Omron Sysmac Studio project Foset_Youtube_jp (Sysmac Studio 1.54.0.64019, StandardProject)

# Controller new_Controller_0: NX102-1220 version 1.48
Units and slaves: Node10 : NX-ECC203 (E001); Unit 1 : NX-PF0630 (N2); Unit 2 : NX-ID4442 (N3); Unit 3 : NX-OD4256 (N4); Unit 4 : NX-ILM400 (N5); Unit 5 : NX-SID800 (N6); Unit 6 : NX-SOD400 (N7)
Task PrimaryTask (priority 4, period or condition 2000): Program0

TYPE Byte2Bool : UNION
    ByteData : BYTE;
    BoolData : ARRAY[0..7] OF bool;
END_UNION END_TYPE
TYPE Byte2Word : UNION
    ByteData : ARRAY[0..1] OF byte;
    WordData : WORD;
END_UNION END_TYPE
TYPE DUT_E3ASHL500MN_ProcessData_Byte3 : STRUCT
    ControlOutput1 : BOOL;
    ControlOutput2 : BOOL;
    LowIntensity : BOOL;
    IssficientLioghtIntensity : BOOL;
    Warning : BOOL;
    Error : BOOL;
END_STRUCT END_TYPE
TYPE DUT_E3ASHL500MN_ProcessData : STRUCT
    DetectionValue : INT;
    LightIntensity : INT;
    Status : DUT_E3ASHL500MN_ProcessData_Byte3;
END_STRUCT END_TYPE

VAR_GLOBAL
    N3_Input_Bit_8_bits : BYTE;  (* at ECAT://node#[10,2]/Input Bit 8 bits *)
    N4_Output_Bit_8_bits : BYTE;  (* at ECAT://node#[10,3]/Output Bit 8 bits *)
    N5_Port2_Input_Data01 : ARRAY[0..1] OF BYTE;  (* at ECAT://node#[10,4]/Port2 Input Data01 *)
    N5_Port2_Input_Data02 : ARRAY[0..1] OF BYTE;  (* at ECAT://node#[10,4]/Port2 Input Data02 *)
    N5_Port2_IN_Data_Enable : BOOL;  (* at ECAT://node#[10,4]/I/O Port Status/Port2 IN Data Enable *)
    N5_IO_Pwr_On : BOOL;  (* at ECAT://node#[10,4]/I/O Port Status/IO Pwr On *)
    N6_Si00_Logical_Value : BOOL;  (* at ECAT://node#[10,5]/Standard Input 1st Word/Si00 Logical Value *)
    N1_DataToSafety_01 : BOOL;  (* at IOBus://unit#1/DataToSafety_01 *)
    N1_DataToSafety_00 : BOOL;  (* at IOBus://unit#1/DataToSafety_00 *)
    N1_Program_Operating : BOOL;  (* at IOBus://unit#1/Program Operating *)
    N1_Program_No_Fault : BOOL;  (* at IOBus://unit#1/Program No Fault *)
    N1_CIP_Safety_Originator_Connection_Status : BOOL;  (* at IOBus://unit#1/CIP Safety Originator Connection Status *)
END_VAR

(* Program Program0: safety or other program stored in binary form, left out *)

PROGRAM Program0
VAR
    NodeReady : BOOL;
    bNoContact : BOOL;
    bNCContact : BOOL;
    MyTimer1 : TON;
    MyTimer2 : TON;
    MyTimer3 : TON;
    MyTimer4 : TON;
    strByte2Bool : Byte2Bool;
    E3AS_1 : FB_E3ASHL500MN;
    Device : DUT_E3ASHL500MN_ProcessData;
    Port2Ready : BOOL;
END_VAR
VAR_EXTERNAL
    N1_DataToSafety_01 : BOOL;
END_VAR
VAR_EXTERNAL CONSTANT
    _EC_MacAdrErr : BOOL;
    _EC_CommErrTbl : ARRAY[1..192] OF BOOL;
END_VAR
VAR_EXTERNAL
    N3_Input_Bit_8_bits : BYTE;
    N1_DataToSafety_00 : BOOL;
    N1_Program_No_Fault : BOOL;
    N1_CIP_Safety_Originator_Connection_Status : BOOL;
    N1_Program_Operating : BOOL;
    N6_Si00_Logical_Value : BOOL;
    N5_Port2_IN_Data_Enable : BOOL;
    N5_IO_Pwr_On : BOOL;
    N5_Port2_Input_Data01 : ARRAY[0..1] OF BYTE;
    N5_Port2_Input_Data02 : ARRAY[0..1] OF BYTE;
    N4_Output_Bit_8_bits : BYTE;
END_VAR
//
	MyTimer3(In:=NOT MyTimer4.Q, PT:=T#0.5s);
	MyTimer4(In:=MyTimer3.Q, PT:=T#0.5s);
	N1_DataToSafety_01:=MyTimer3.Q;
	
//
	NodeReady:=_EC_MacAdrErr = 0 AND NOT _EC_CommErrTbl[2];
	strByte2Bool.ByteData:=0;
	strByte2Bool.ByteData:=N3_Input_Bit_8_bits;
	bNoContact:=strByte2Bool.BoolData[0];
	bNCContact:=strByte2Bool.BoolData[1];
	N1_DataToSafety_00:=strByte2Bool.BoolData[2] AND 
			N1_Program_No_Fault AND N1_Program_Operating AND N6_Si00_Logical_Value;
//
	strByte2Bool.ByteData:=0;
	NodeReady:=_EC_MacAdrErr = 0 AND NOT _EC_CommErrTbl[3];
	MyTimer1(In:=bNoContact AND NOT MyTimer2.Q, PT:=T#1s);
	MyTimer2(In:=MyTimer1.Q, PT:=T#1s);
	strByte2Bool.BoolData[1]:=bNCContact OR MyTimer1.Q;
	N4_Output_Bit_8_bits:=strByte2Bool.ByteData;
	
//
	Port2Ready:=N5_Port2_IN_Data_Enable AND N5_IO_Pwr_On;
	NodeReady:=_EC_MacAdrErr = 0 AND NOT _EC_CommErrTbl[5];
	E3AS_1	(IoData1:=N5_Port2_Input_Data01,IoData2:=N5_Port2_Input_Data02
				,ioE3AS:=Device
				);
				
END_PROGRAM

FUNCTION_BLOCK FB_E3ASHL500MN
VAR
    Temp : BOOL;
    uByte2Word : Byte2Word;
    uByteBool : Byte2Bool;
END_VAR
VAR_IN_OUT
    ioData1 : ARRAY[0..1] OF byte;
    ioData2 : ARRAY[0..1] OF byte;
    ioE3AS : DUT_E3ASHL500MN_ProcessData;
END_VAR
//

Temp:=TRUE;

uByte2Word.ByteData[0]:=ioData1[1];
uByte2Word.ByteData[1]:=ioData1[0];

ioE3AS.DetectionValue:=WORD_TO_INT(uByte2Word.WordData);
ioE3AS.LightIntensity:=BYTE_TO_INT(ioData2[0]);

uByteBool.ByteData:=ioData2[1];

ioE3AS.Status.ControlOutput1:=uByteBool.BoolData[0];
ioE3AS.Status.ControlOutput2:=uByteBool.BoolData[1];
ioE3AS.Status.LowIntensity:=uByteBool.BoolData[2];
ioE3AS.Status.IssficientLioghtIntensity:=uByteBool.BoolData[4];
ioE3AS.Status.Warning:=uByteBool.BoolData[6];
ioE3AS.Status.Error:=uByteBool.BoolData[7];
END_FUNCTION_BLOCK